FUNCTION_BLOCK FB_Syntax_VarInOut VAR_INPUT nFactor : INT := 1; END_VAR VAR_IN_OUT nCounter : INT; END_VAR VAR _stLocal  : ST_Syntax_Mini; _nScratch : INT; END_VAR

_nScratch      := nCounter * nFactor;
nCounter       := _nScratch;
_stLocal.nId   := nCounter;
_stLocal.sName := 'Updated';

METHOD M_Process : INT VAR_INPUT nDelta : INT; END_VAR VAR_INST _nInstanceCounter : INT; END_VAR
_nInstanceCounter := _nInstanceCounter + nDelta;
M_Process         := _nInstanceCounter;
END_METHOD

END_FUNCTION_BLOCK

(* stored: Version 1.1.0.1, ProductVersion 3.1.4024.16
   POU FB_Syntax_VarInOut: Id {d14581f1-1e3d-4b96-964c-55be4b83bf4d}, SpecialFunc None
   Method M_Process: Id {c5793e1a-4d2a-43cf-8a03-7f12e9b87b21} *)
